// SIMATIC S7-200 SMART project (STEP 7-Micro/WIN SMART), CPU CR40

SYMBOL_TABLE 系统符号
Clock_1s         SM0.5    // 针对 1 s 的周期时间，时钟脉冲接通 0.5 s，断开 0.5 s.
END_SYMBOL_TABLE

ORGANIZATION_BLOCK MAIN:OB1
TITLE=M0.0：故障状态
// M0.1：急停状态
// M1.0：工作状态
BEGIN
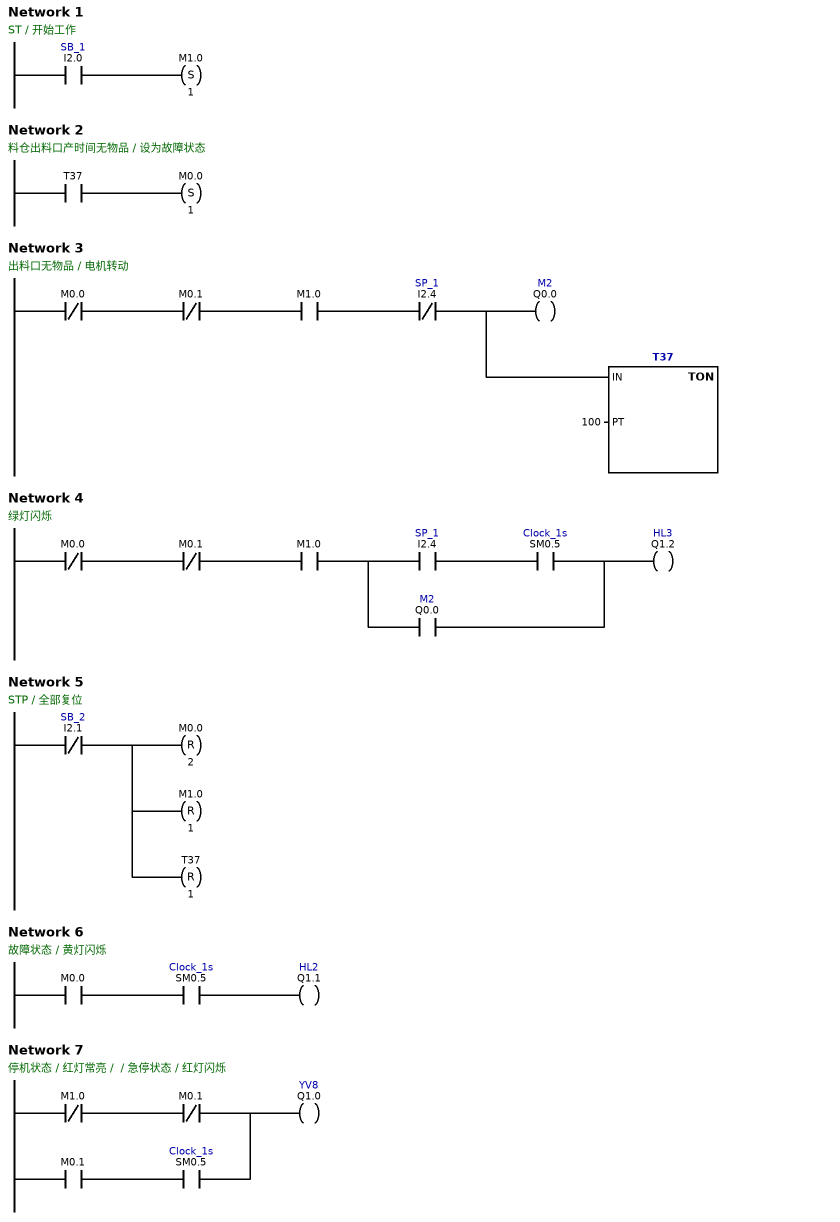
Network 1
// ST
// 开始工作
LD     SB_1:I2.0
S      M1.0, 1
Network 2
// 料仓出料口产时间无物品
// 设为故障状态
LD     T37
S      M0.0, 1
Network 3
// 出料口无物品
// 电机转动
LDN    M0.0
AN     M0.1
A      M1.0
AN     SP_1:I2.4
=      M2:Q0.0
TON    T37, 100
Network 4
// 绿灯闪烁
LDN    M0.0
AN     M0.1
A      M1.0
LD     SP_1:I2.4
A      Clock_1s:SM0.5
O      M2:Q0.0
ALD
=      HL3:Q1.2
Network 5
// STP
// 全部复位
LDN    SB_2:I2.1
R      M0.0, 2
R      M1.0, 1
R      T37, 1
Network 6
// 故障状态
// 黄灯闪烁
LD     M0.0
A      Clock_1s:SM0.5
=      HL2:Q1.1
Network 7
// 停机状态
// 红灯常亮
// 
// 急停状态
// 红灯闪烁
LDN    M1.0
AN     M0.1
LD     M0.1
A      Clock_1s:SM0.5
OLD
=      YV8:Q1.0
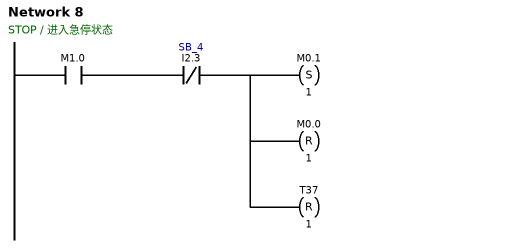
Network 8
// STOP
// 进入急停状态
LD     M1.0
AN     SB_4:I2.3
S      M0.1, 1
R      M0.0, 1
R      T37, 1
END_ORGANIZATION_BLOCK
